// TIA Portal V19 export
FUNCTION "A0302_Bordatrice_CALL" : Void   // FC181, LAD
TITLE = << BORDATRICE MOVIMENTO >>
// stored: SetENOAutomatically false
   VAR CONSTANT
      MinimumPos : Real := 0.0;
      MaximumPos : Real := 1000.0;
      MISSING : Int;
   END_VAR
BEGIN

REGION Network 1 (SCL): << TRASFERIMENTO stati CIn del blocco >>
   // SOSTITUIRE SYS BYPASS CON INGRESSI DIGITALI

   // TRASFERIMENTO COMANDI CIn MANAGER
   "A0302_Bordatrice".CIn.Manager.Ax := "A0302_Manager".COut.Bordatrice.Ax;
   //
   "A0302_Bordatrice".CIn.SemiAut_Pb := "A0302_Manager".DataIn.SemiAut_Pb;


   REGION TRASFERIMENTO CIn DIGITAL INPUT dei LIMIT SWITCH
       //
       //"A0302_Bordatrice".Ax.CIn.PositionLimits.EnableMin := FALSE;
       //"A0302_Bordatrice".Ax.CIn.PositionLimits.EnableMax := FALSE;

   END_REGION ;

   REGION TRASFERIMENTO STATI STAZIONE P5

       "A0302_Bordatrice".CIn.P5.Sollevatori := "A0301_Spintore_Lat".COut.Sollevatori;
       "A0302_Bordatrice".CIn.P5.SpintoreLong := "A0302_Spintore".COut.Spintore;
       "A0302_Bordatrice".CIn.P5.Sens.FTC_Ingombro_A0301 := "A0302_Spintore".IEC.FTC_On;

   END_REGION ;

   REGION  TRASFERIMENTO STATI RULLIERA dopo BORDATRICE

       "A0302_Bordatrice".CIn.Rulliera.Centratori := "A0302_Centratori".COut.Centraggio;
       "A0302_Bordatrice".CIn.Rulliera.Sollevatori := "A0302_Centratori".COut.Sollevamento;
       "A0302_Bordatrice".CIn.Rulliera.Coda.Sens := "A0302_Manager".CIn.Rulliera.Coda.Sens;
       "A0302_Bordatrice".CIn.Rulliera.Centro.Sens := "A0302_Manager".CIn.Rulliera.Centro.Sens;

   END_REGION ;

   REGION TRASFERIMENTO STATI CARRO PAREGGIATORE DI CODA

       "A0302_Bordatrice".CIn.CarroPareggCoda.Ax := "A0302_PareggiatoreCoda".COut.Ax;
       "A0302_Bordatrice".CIn.CarroPareggCoda.Bloccaggio := "A0302_PareggiatoreCoda".COut.Bloccaggio;
       "A0302_Bordatrice".CIn.CarroPareggCoda.BattutaVerticale := "A0302_PareggiatoreCoda".COut.BattutaVerticale;
       "A0302_Bordatrice".CIn.CarroPareggCoda.PareggiatoreLongitudinale := "A0302_PareggiatoreCoda".COut.PareggiatoreLong;
       "A0302_Bordatrice".CIn.CarroPareggCoda.Sens := "A0302_Manager".CIn.CarroPareggCoda.Sens;

   END_REGION ;

   REGION  TRASFERIMENTO STATI CARRO PAREGGIATORE DI TESTA

       "A0302_Bordatrice".CIn.CarroPareggTesta.Ax := "A0302_PareggiatoreTesta".COut.Ax;
       "A0302_Bordatrice".CIn.CarroPareggTesta.Bloccaggio := "A0302_PareggiatoreTesta".COut.Bloccaggio;
       "A0302_Bordatrice".CIn.CarroPareggTesta.Centraggio := "A0302_PareggiatoreTesta".COut.Centraggio;
       "A0302_Bordatrice".CIn.CarroPareggTesta.Sollevatore := "A0302_PareggiatoreTesta".COut.Sollevatore;
       "A0302_Bordatrice".CIn.CarroPareggTesta.Sens := "A0302_Manager".CIn.CarroPareggTesta.Sens;

   END_REGION ;

   // ATTREZZAGGIO PRONTO
   "A0302_Bordatrice".CIn.Attrezzaggio.CarriParegg.Ready := "A0302_Manager".Sts.Attrezzamento.Ready;
END_REGION

REGION Network 2 (SCL): << TRASFERIMENTO stati DataIn >>
   REGION TRASFERIMENTO #DataIn STATI BUTTON BORDATRICE
       // PB BORDATRICE
       "A0302_Bordatrice".Ax.DataIn.PB.Bwd_Minus := "A03_HMI".MB3.Button.A0302.Bordatrice.Ax.Bwd_Minus;
       "A0302_Bordatrice".Ax.DataIn.PB.Fwd_Plus := "A03_HMI".MB3.Button.A0302.Bordatrice.Ax.Fwd_Plus;
       "A0302_Bordatrice".Ax.DataIn.PB.MoveToPos := "A03_HMI".MB3.Button.A0302.Bordatrice.Ax.MoveToPos;

       // Sensori
       "A0302_Bordatrice".DataIn.Sens.FTC_Uscita := "A0302_Bordatrice_Banco_4_Lato_1_Phc_AtExit";

       // Feedback connettori
       "A0302_Bordatrice".DataIn.FdBack.ConnMotori := "A0302_Bordatrice_ControlloConnettoreBanco_4_Lato_1";
       "A0302_Bordatrice".DataIn.FdBack.ConnAux := "A0302_Bordatrice_ControlloConnettoreBanco_4_Lato_2";

   END_REGION ;
END_REGION

REGION Network 3 (SCL): DSI
   //
   "A0302_Bordatrice".DSI := "F_DB".DSI_S120_Bordatrice;
END_REGION

REGION Network 4 (SCL): HW
   //
   "A0302_Bordatrice".HWID_TEL111 := "HW_Const_Values".CU5_PN_1950A1_SIEMENS_telegram_111;
END_REGION

REGION Network 5 (SCL): Drive
   //
   "A0302_Bordatrice".Drive.Infeed_ON := "Areas_ITF".AG.Infeed_Running;
   "A0302_Bordatrice".Drive.AccessPoint := "HW_Const_Values".CU5_PN_1950A1_ModuleAccessPoint;
   "A0302_Bordatrice".Drive.AxisID := "CU5_ID_2_1950A1_1950M1";
   "A0302_Bordatrice".Drive.TokenChain := "TOKENCHAIN_CU5";
END_REGION

REGION Network 6: [Bordatrice] - Machine call
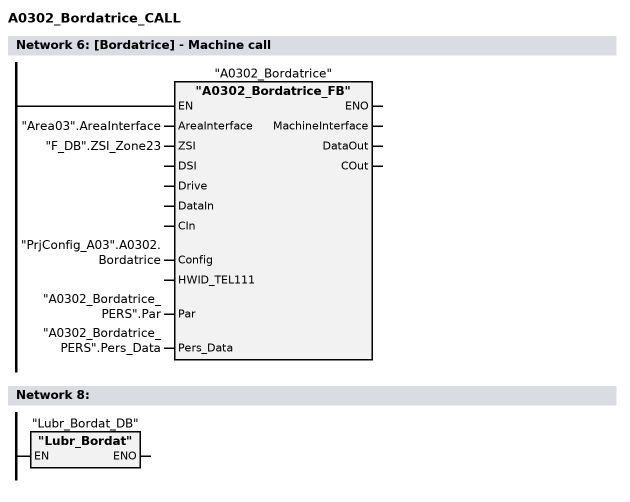
   RUNG wire#powerrail
      "A0302_Bordatrice"(AreaInterface := "Area03".AreaInterface, ZSI := "F_DB".ZSI_Zone23, DSI :=, Drive :=, DataIn :=, CIn :=, Config := "PrjConfig_A03".A0302.Bordatrice, HWID_TEL111 :=, Par := "A0302_Bordatrice_PERS".Par, Pers_Data := "A0302_Bordatrice_PERS".Pers_Data, MachineInterface =>, DataOut =>, COut =>)
   END_RUNG
   // the same network as SCL:
   "A0302_Bordatrice"(AreaInterface := "Area03".AreaInterface,   // "A0302_Bordatrice_FB"
                      ZSI := "F_DB".ZSI_Zone23,
                      Config := "PrjConfig_A03".A0302.Bordatrice,
                      Par := "A0302_Bordatrice_PERS".Par,
                      Pers_Data := "A0302_Bordatrice_PERS".Pers_Data);
END_REGION

REGION Network 8
   RUNG wire#powerrail
      "Lubr_Bordat_DB"()
   END_RUNG
   // the same network as SCL:
   "Lubr_Bordat_DB"();   // "Lubr_Bordat"
END_REGION
END_FUNCTION
